# EPICS autosave request: stdApp/Db/scanParms_settings.req
# FILE... scanParms_settings.req
# USAGE.. scanParms.db fields autosave'd.
$(P)$(M):scanParms.SP
$(P)$(M):scanParms.EP
$(P)$(M):scanParms.NP
$(P)$(M):scanParms.AR
$(P)$(M):scanParms.AFT
